Omron CX-Programmer project NewProject (CX-Programmer 9.70)

# PLC NewPLC1: CP1E E20

## Global symbols (name address type ; comment)
0.01 BOOL  ; START
0.04 BOOL  ; STOP
100.00 BOOL  ; LED

## Program NewProgram1 (cyclic task 0)

### Section Section1

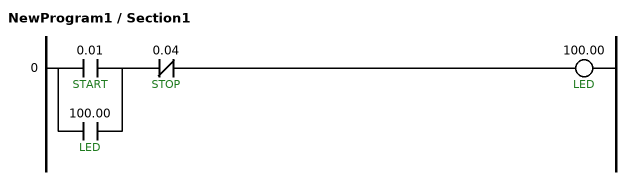
; rung 0
LD 0.01  ; START
OR 100.00  ; LED
ANDNOT 0.04  ; STOP
OUT 100.00  ; LED

### Section END
; rung 0
END(001)